Yaskawa INFORM job: SENSORES.JBI

/JOB
//NAME SENSORES
///FOLDERNAME SENSORES
//POS
///NPOS 0,0,0,0,0,0
//INST
///DATE 2022/06/04 11:52
///ATTR SC,RW
NOP
'VERIFICACAO SENSORES OFF
WAIT IN#(549)=OFF
WAIT IN#(550)=OFF
END
